// TwinCAT 3 PLC project Temp_PID_cascade
// ProgramVersion: 3.1.4023.0
// libraries:
//   Tc2_ControllerToolbox,3.4.1.4,Beckhoff Automation GmbH
//   Tc2_Math,3.3.1.0,Beckhoff Automation GmbH
//   Tc2_Standard,3.3.3.0,Beckhoff Automation GmbH
//   Tc2_System,3.4.22.0,Beckhoff Automation GmbH
//   Tc2_TempController,3.3.4.0,Beckhoff Automation GmbH
//   Tc3_Module,3.3.21.0,Beckhoff Automation GmbH
// project tree:
//   GVLs/ gbl.TcGVL, IOgbl.TcGVL
//   / PlcTask.TcTTO
//   POUs/ MAIN.TcPOU, master.TcPOU, slave.TcPOU
// real-time tasks:
//   TASK PlcTask: cycle T#1ms, priority 20, ADS port 350
// I/O:
//   DEVICE Device 1 (EtherCAT) (disabled), AmsNetId 192.168.56.1.2.1
//     Term 1 (EK1200) [EK1200-5000 EtherCAT Power supply (2A E-Bus)]
//       Term 2 (EL3318) [EL3318 8Ch. Ana Input Thermocouple (TC)]
//       Term 3 (EL3318) [EL3318 8Ch. Ana Input Thermocouple (TC)]
//       Term 4 (EL4024) [EL4024 4Ch. Ana. Output 4-20mA, 12bit]
//       Term 5 (EL9011) [EL9011 End Terminal]
// variable links:
//   Temp_PID_cascade/Temp_PID_cascade Instance <-> Device 1 (EtherCAT)/Term 1 (EK1200)/Term 2 (EL3318)
//     PlcTask Inputs/IOgbl.AI_IO_ST_temp[1] <-> TC Channel 8/Value
//     PlcTask Inputs/IOgbl.AI_IO_slave_pv[{1..4}] <-> TC Channel {1..4}/Value  (4 links)
//   Temp_PID_cascade/Temp_PID_cascade Instance <-> Device 1 (EtherCAT)/Term 1 (EK1200)/Term 3 (EL3318)
//     PlcTask Inputs/IOgbl.AI_IO_ST_temp[{2..9}] <-> TC Channel {1..8}/Value  (8 links)
//   Temp_PID_cascade/Temp_PID_cascade Instance <-> Device 1 (EtherCAT)/Term 1 (EK1200)/Term 4 (EL4024)
//     PlcTask Outputs/IOgbl.AO_IO_SCR_set[{1..4}] <-> AO Outputs Channel {1..4}/Analog output  (4 links)

CONFIGURATION Temp_PID_cascade
    RESOURCE PLC ON TwinCAT3
        TASK PlcTask(INTERVAL := T#1ms, PRIORITY := 20);
        PROGRAM MAIN WITH PlcTask : MAIN;
    END_RESOURCE
END_CONFIGURATION

// ---- GVLs/gbl.TcGVL
{attribute 'qualified_only'}
VAR_GLOBAL
	(*===========================================main=====================================*)
	bWatch						 : BOOL;
	tuning_mode 	     		 : BOOL;
	tuning_time	     			 : LREAL;
	tune_result					 :  ARRAY[1..4] OF LREAL;
	
	(*===========================================master====================================*)
	master_bRamp_Enable          : BOOL;
	(*---------------------input------------------------*)
	master_fRamp_Value           : ARRAY[1..4] OF LREAL := [10, 10, 10, 10] ;
	master_TargetTemp            : LREAL;
	master_pi_gain               : ARRAY[1..4] OF LREAL;	//PI제어기 이득(gain) -P
	master_integral_constant	 : ARRAY[1..4] OF LREAL;	//PI제어기 적분상수 -I
	master_Zone_Temp_Min         : LREAL;  //단위 : %
	master_Zone_Temp_Max         : LREAL;  //단위 : %
	
	(*===========================================sub TC===================================*)
	(*---------------------output------------------------*)
	fPV_Value_SubTC				: ARRAY[1..9] OF LREAL; (* glass 각각의 온도 *)
	subTC_max 					: LREAL ;
	subTC_min 					: LREAL ;
	subTC_dev					: LREAL ;  (* glss_max - glass_min *)
	subTC_AVG                   : LREAL ;  (* glass temp AVG *)
	
	(*=======================================slave========================================*)	
	slave_bsimulation		   : BOOL;
	slave_bRamp_Enable         : ARRAY[1..4] OF BOOL;
	(*---------------------input------------------------*)
	slave_fRamp_Value          : ARRAY[1..4] OF LREAL ;
	slave_fTargetTemp          : ARRAY[1..4] OF LREAL ;
	slave_fPowLimit            : ARRAY[1..4] OF LREAL ;
	slave_eCTRL_MODE           : ARRAY[1..4] OF E_CTRL_MODE ;
	slave_bstart			   : BOOL ;

	slave_fP_Value	           : ARRAY[1..4] OF LREAL  ;
	slave_tI_Value		       : ARRAY[1..4] OF LREAL  ;
	slave_tD_Value		       : ARRAY[1..4] OF LREAL  ;
	slave_bEmergency_Stop	   : BOOL ;
	(*---------------------output------------------------*)
	slave_fPV_Value				: ARRAY[1..4] OF LREAL;
	slave_fMV_Out				: ARRAY[1..4] OF LREAL;
	slave_fRamp_Out 		    : ARRAY[1..4] OF LREAL;
	slave_nErrorID			    : E_CTRL_ERRORCODES;	
	slave_bError				: BOOL;
END_VAR

// ---- GVLs/IOgbl.TcGVL
{attribute 'qualified_only'}
VAR_GLOBAL
	AI_IO_slave_pv  AT%IB1001   :   ARRAY [1..4] OF UINT;
	AI_IO_ST_temp   AT%IB1021   :   ARRAY [1..9] OF UINT;
	
	
	AO_IO_SCR_set 	AT%QB1051 	:   ARRAY [1..4] OF UINT;  
END_VAR

// ---- POUs/MAIN.TcPOU
PROGRAM MAIN
VAR	
	onTimer 			: TON;
	OffTimer 			: TOF;
	timerStart			: BOOL;
	reverseSignal 		: BOOL;
	
	onTimer_tune  		: TON;
	OffTimer_tune 		: TOF;
	reverseSignal_tune  : BOOL;
	
	i    				: INT;

END_VAR


IF gbl.slave_bsimulation = FALSE THEN

	FOR i:=1 TO 4 BY 1 DO
		gbl.slave_fPV_Value[i] := IOgbl.AI_IO_slave_pv[i] / 10 ;
		IOgbl.AO_IO_SCR_set[i] := LREAL_TO_UINT(gbl.slave_fMV_Out[i] * 327.67);
	END_FOR
	
	FOR i:=1 TO 9 BY 1 DO
		gbl.fPV_Value_SubTC[i] := IOgbl.AI_IO_ST_temp[i] / 10 ;
	END_FOR
	
ELSE
	slave.SIMULATION() ;
END_IF

(* watch dogs : 10s 간격으로 on/ off *)
onTimer(IN := OffTimer.Q, PT := T#10S);
IF onTimer.Q THEN
  reverseSignal := FALSE;
  gbl.bWatch := FALSE;
ELSE
  reverseSignal := TRUE;
  gbl.bWatch := TRUE;
END_IF
OffTimer(IN := reverseSignal, PT := T#10S);

(* 
mgbl.master_tuning_mode = tune set
tune set :  true -> master, slave호출
tune set :  false -> slave만 호출
*)
IF gbl.tuning_mode THEN

	master();
	slave();
	
  (* 튜닝 시간 설정 = mgbl.master_tuning_time *)
    onTimer_tune(IN := OffTimer_tune.Q, PT := LREAL_TO_TIME(gbl.tuning_time)*60000); // IN이 FALSE에서 TRUE가 되자마자 시간이 흐름,PT와 같아지면 Q가 TRUE
    IF onTimer_tune.Q THEN
	  gbl.tuning_mode := FALSE;
	  reverseSignal_tune := FALSE;
	  gbl.tune_result := gbl.slave_fPV_Value;
	ELSE
	  reverseSignal_tune := TRUE;
    END_IF
    OffTimer_tune(IN := reverseSignal_tune, PT := T#0S); // IN이 TRUE에서 FALSE가 되자마자 시간이 흐름, PT와 같아지면 Q가 FALSE
	FOR i:=1 TO 4 BY 1 DO
		gbl.tune_result[i] := 0;
	END_FOR
ELSE
	slave();
END_IF

END_PROGRAM

// ---- POUs/slave.TcPOU
PROGRAM slave
VAR
	fPV_Value_					:			ARRAY[1..4] OF LREAL ;
	
	tTime						:			TIME ;
	tTaskCycleTime				:			TIME := T#1MS ;
	tCtrlCycleTime				:			TIME := T#200MS ;
	
	fbCTRL_PT2				    : 			ARRAY[1..4] OF FB_CTRL_PT2 ;
	stPTParams				    : 			ARRAY[1..4] OF ST_CTRL_PT2_PARAMS ;

	stCTRL_ParaController_Ex	:			ARRAY[1..4] OF ST_CTRL_ParaController ;
	stCTRL_ParaController_In	:			ARRAY[1..4] OF ST_CTRL_ParaController ;
	stCTRL_TempCtrlParameter	:			ARRAY[1..4] OF ST_CTRL_TempCtrlParameter ;
	
	fbCTRL_TempController		:			ARRAY[1..4] OF FB_CTRL_TempController ;
		
	eCTRL_STATE					:			ARRAY[1..4] OF E_CTRL_STATE ;
	
	e_Heat_Mode					:			E_CTRL_ControlMode 			:= eCTRL_ControlMode_HEATING ;
	e_Fail_Action				:			E_CTRL_ReactionOnFailure 	:= eCTRL_ReactionOnFailure_NoFailure ;
		
	s_bError					:			BOOL ;
	s_nErrorID					:			E_CTRL_ERRORCODES ;
	s_fMaxOvershoot				:			LREAL ;
	
	s_bFirst					:			BOOL := TRUE ;
	
	(* Ramp Parameter Set *)
	s_bRamp_Use				    :			ARRAY[1..4] OF BOOL ;	
	s_fRamp_Rate				:			ARRAY[1..4] OF LREAL ;
	
	(* =============== Setting Item 입력 =============== *)
	
	(* PID Set Parameter *)
	s_fP_Value						:			ARRAY[1..4] OF LREAL ;
	s_tI_Value						:			ARRAY[1..4] OF TIME	;
	s_tD_Value						:			ARRAY[1..4] OF TIME	;
	
	(* Power Limit Set *)
	s_fPowLimit					:			ARRAY[1..4] OF LREAL ;
	
	(* Manual Control 시 Power 출력값 *)
	s_fSetManual					:			ARRAY[1..4] OF LREAL ;
	
	(*	Heater Mode	*)
	s_eCTRL_MODE					:			ARRAY[1..4] OF E_CTRL_MODE ;			(* Auto Mode 동작은 2 : eCTRL_MODE_ACTIVE 설정 *)
	
	(*	온도 설정 입력	*)
	s_fSet_Value					:			ARRAY[1..4] OF LREAL ;
	s_fLast_Set_Value            	:           ARRAY[1..4] OF LREAL ;

	
	(*	비상정지	*)
	//bEmergency_Stop					:			ARRAY[1..4] OF BOOL ;
	
	fbCTRL_RAMP_GENERATOR			 :   ARRAY[1..4] OF FB_CTRL_RAMP_GENERATOR ;
	stCTRL_RAMP_GENERATOR_PARAMS     :   ARRAY[1..4] OF ST_CTRL_RAMP_GENERATOR_PARAMS ;
	
	System_step	: INT ;
	
	i    :   INT ;
	
	master_Zone_AVG	                 :   ARRAY[1..4] OF LREAL ;
	
END_VAR

(* ================ Simulation Constant Parameter =======================*)
VAR CONSTANT
	fKp							:			ARRAY[1..4] OF REAL := [15.5, 15.2, 15.7, 15.8] ;
	fInit_Temp					:			ARRAY[1..4] OF REAL := [23.5, 23.8, 23.9, 23.7] ;
	tTimeConstant				:			ARRAY[1..4] OF TIME := [T#251.4S, T#252.4S, T#254.4S, T#256.4S] ;
END_VAR

(*
IF gbl.slave_bsimulation THEN
   SIMULATION();
END_IF
*)

IF gbl.slave_bError THEN
   gbl.slave_bEmergency_Stop := TRUE ;
END_IF

FOR i:=1 TO 4 BY 1 DO
   IF gbl.slave_bEmergency_Stop THEN
      s_fSet_Value[i] := 0;
      s_fPowLimit[i] := 0;
      s_eCTRL_MODE[i] := eCTRL_MODE_IDLE;
      fbCTRL_TempController[i]( eCtrlMode := s_eCTRL_MODE[i],      
              bSelSetpoint            := FALSE,
              fw1                     := s_fSet_Value[i],
              fw2                     := ,            
              fX                      := gbl.slave_fPV_Value[i],      
              fyManual                := s_fSetManual[i],
              sParaControllerExternal := stCTRL_ParaController_Ex[i],
              sControllerParameter    := stCTRL_TempCtrlParameter[i]
              );
   ELSE
      s_fPowLimit[i] := gbl.slave_fPowLimit[i];
      s_eCTRL_MODE[i] := gbl.slave_eCTRL_MODE[i];
   END_IF
END_FOR

IF s_bFirst THEN
   DEFAULT_PARA_SET();
   s_bFirst := FALSE ;
   System_step :=0;
END_IF

CASE System_step OF
      
   0:

      s_bRamp_Use     :=  gbl.slave_bRamp_Enable;
      s_fRamp_Rate    :=  gbl.slave_fRamp_Value;
	  
      IF gbl.slave_bStart THEN
         FOR i:=1 TO 4 BY 1 DO
            s_fLast_Set_Value[i] := s_fSet_Value[i];
         END_FOR
         FOR i:=1 TO 4 BY 1 DO
            s_fSet_Value[i] := gbl.slave_fTargetTemp[i];
         END_FOR
         System_step := 1;
         gbl.slave_bStart := FALSE;
         ELSE
            System_step := 0;
      END_IF
      

   1:
      FOR i:=1 TO 4 BY 1 DO
         s_fP_Value[i] := gbl.slave_fP_Value[i];
         s_tI_Value[i] := LREAL_TO_TIME(gbl.slave_tI_Value[i]);
         s_tD_Value[i] := LREAL_TO_TIME(gbl.slave_tD_Value[i]);
         
         IF s_fP_Value[i] <= 0 THEN
            s_fP_Value[i] := 0.1;
         ELSE
            s_fP_Value[i] := s_fP_Value[i];
         END_IF

         stCTRL_ParaController_Ex[i].KpHeat := s_fP_Value[i];   
         stCTRL_ParaController_Ex[i].TnHeat := s_tI_Value[i];
         stCTRL_ParaController_Ex[i].TvHeat := s_tD_Value[i];
         stCTRL_ParaController_Ex[i].TdHeat := T#1S;
         
         System_step := 2;
         
      END_FOR
      
      System_step := 2;

   2:
      
      FOR i:=1 TO 4 BY 1 DO
         IF s_fPowLimit[i] > 100 THEN
            s_fPowLimit[i] := 100;
         ELSE 
            s_fPowLimit[i] := s_fPowLimit[i];
         END_IF
      
         stCTRL_TempCtrlParameter[i].fYMax := s_fPowLimit[i];
         
         stCTRL_RAMP_GENERATOR_PARAMS[i].fVeloNeg := s_fRamp_Rate[i] / 60.0;
         stCTRL_RAMP_GENERATOR_PARAMS[i].fVeloPos := s_fRamp_Rate[i] / 60.0;
         
         System_step := 3;
      
      END_FOR
       
      System_step := 3;
   
   3:
      
      FOR i:=1 TO 4 BY 1 DO
      
         IF s_fSetManual[i] > 100 THEN
            s_fSetManual[i] := 100;
         ELSE
            s_fSetManual := s_fSetManual;
         END_IF

         stCTRL_TempCtrlParameter[i].fYManual         :=   s_fSetManual[i];          
         stCTRL_TempCtrlParameter[i].fYOnFailure      :=   s_fSet_Value[i];
      END_FOR
      
      System_step := 4;
     
   4:
      FOR i:=1 TO 4 BY 1 DO
         fbCTRL_TempController[i]( eCtrlMode               := gbl.slave_eCTRL_MODE[i],      
                             bSelSetpoint            := FALSE,
                             fw1                     := s_fSet_Value[i],
                             fw2                     := ,            
                             fX                      := gbl.slave_fPV_Value[i],      
                             fyManual                := s_fSetManual[i],
                             sParaControllerExternal := stCTRL_ParaController_Ex[i],
                             sControllerParameter    := stCTRL_TempCtrlParameter[i]
                             );
        END_FOR
      
      System_step := 100;
      
   100:
      System_step := 0;
      
END_CASE


Ramping();

FOR i:=1 TO 4 BY 1 DO 
   
   fbCTRL_TempController[i](
                 fw1                       := gbl.slave_fRamp_Out[i],
                 fX                        := gbl.slave_fPV_Value[i],    
                 sParaControllerExternal   := stCTRL_ParaController_Ex[i],
                 sControllerParameter      := stCTRL_TempCtrlParameter[i],
                 fYAnalog                   => gbl.slave_fMV_Out[i],
                 bYPWMPos                   => ,
                 bYPWMNeg                   => ,
                 dwAlarm                    => ,
                 fMaxOverShoot              => s_fMaxOvershoot,
                 tStartUpTime               => ,
                 eCtrlState                 => eCTRL_STATE[i],
                 sParaControllerInternal    => stCTRL_ParaController_In[i],
                 bError                     => gbl.slave_bError,
                 eErrorId                   => gbl.slave_nErrorID
                );
END_FOR

ACTION DEFAULT_PARA_SET:
FOR i := 1 TO 4 DO
	stCTRL_TempCtrlParameter[i].iMode				:=	e_Heat_Mode;
	stCTRL_TempCtrlParameter[i].iReactionOnFailure  :=	e_Fail_Action;
	stCTRL_TempCtrlParameter[i].dwAlarmSupp		    :=	16#FF_FF_FF_FF;		(* alarm suppression  Default 사용 *)
	stCTRL_TempCtrlParameter[i].fWMin				:=	0.0;
	stCTRL_TempCtrlParameter[i].fWMax				:=	500;
	stCTRL_TempCtrlParameter[i].bEnableSoftStart	:=	FALSE;
	stCTRL_TempCtrlParameter[i].fWStartUp			:=	30.0;
	stCTRL_TempCtrlParameter[i].tStartUp			:=	T#1S;
	stCTRL_TempCtrlParameter[i].bStartUpRamping	    :=	FALSE;
	stCTRL_TempCtrlParameter[i].fWStartUpVeloPos	:=	0.1;
	stCTRL_TempCtrlParameter[i].fWStartUpVeloNeg	:=	0.1;
	stCTRL_TempCtrlParameter[i].bFilter			    :=	FALSE;
	stCTRL_TempCtrlParameter[i].tFilter			    :=	T#0S;
	stCTRL_TempCtrlParameter[i].bDeadband			:=	FALSE;
	stCTRL_TempCtrlParameter[i].fEDeadband			:=	0.0;
	stCTRL_TempCtrlParameter[i].tPWMCycleTime		:=	T#1S;
	stCTRL_TempCtrlParameter[i].tPWMMinOffTime		:=	T#0S;
	stCTRL_TempCtrlParameter[i].tPWMMinOnTime		:=	T#0S;
	stCTRL_TempCtrlParameter[i].tPWMWaitingTime	    :=	T#0S;
	stCTRL_TempCtrlParameter[i].fYThresholdOff		:=	0.0;
	stCTRL_TempCtrlParameter[i].fYThresholdOn		:=	0.0;
	stCTRL_TempCtrlParameter[i].TempLow			    :=	-10.0;
	stCTRL_TempCtrlParameter[i].TempLowLow			:=	-5.0;
	stCTRL_TempCtrlParameter[i].TempHigh			:=	5.0;
	stCTRL_TempCtrlParameter[i].TempHighHigh		:=	10.0;
	stCTRL_TempCtrlParameter[i].TempAbsoluteHigh	:=	300.0;
	stCTRL_TempCtrlParameter[i].TempAbsoluteLow	    :=	0.0;
	stCTRL_TempCtrlParameter[i].tCtrlCycleTime		:= 	tCtrlCycleTime;
	stCTRL_TempCtrlParameter[i].tTaskCycleTime		:= 	tTaskCycleTime;
	stCTRL_TempCtrlParameter[i].fYMin				:=	0.0;
	stCTRL_TempCtrlParameter[i].iControllerType	    := eCTRL_ControllerType_PID;
	stCTRL_TempCtrlParameter[i].iFilterType		    := eCTRL_FilterType_FIRSTORDER;
	stCTRL_TempCtrlParameter[i].bEnablePreController:= FALSE;
	stCTRL_TempCtrlParameter[i].bEnableZones 		:= FALSE;
	stCTRL_TempCtrlParameter[i].bEnableCVFilter     := FALSE;
	
	stCTRL_TempCtrlParameter[i].bSelCtrlParameterSet := TRUE;
	
	stCTRL_RAMP_GENERATOR_PARAMS[i].tCtrlCycleTime		:= 	tCtrlCycleTime;
	stCTRL_RAMP_GENERATOR_PARAMS[i].tTaskCycleTime		:= 	tTaskCycleTime;
END_FOR
END_ACTION

ACTION RAMPING:

;
FOR i:=1 TO 4 BY 1 DO
	IF s_bRamp_Use[i] THEN

		fbCTRL_RAMP_GENERATOR[i]( bEnable   := s_bRamp_Use[i],
								fStart   := s_fLast_Set_Value[i],
								fTarget  := s_fSet_Value[i],
								stParams := stCTRL_RAMP_GENERATOR_PARAMS[i],
								fOut   => gbl.slave_fRamp_Out[i],
								fVeloOut  => ,
								bValueReached => ,
								eErrorId => ,
								bError =>
								)
	;			

	ELSE
			gbl.slave_fRamp_Out[i] := s_fSet_Value[i];
		;
	END_IF
END_FOR
END_ACTION

ACTION SIMULATION:


FOR i:=1 TO 4 BY 1 DO
	stPTParams[i].tTaskCycleTime	:= tTaskCycleTime;
	stPTParams[i].tCtrlCycleTime	:= tCtrlCycleTime;
	stPTParams[i].tT1				:= stPTParams[i].tT2 := tTimeConstant[i];
	stPTParams[i].fKp				:= fKp[i];


	fbCTRL_PT2[i](
					fIn			:= gbl.slave_fMV_Out[i] ,
					eMode		:= eCtrl_MODE_ACTIVE,
					stParams	:= stPTParams[i],
					fOut		=> fPV_Value_[i]
					);	
					
	IF fPV_Value_[i] <= fInit_Temp[i] THEN
		gbl.slave_fPV_Value[i] := fInit_Temp[i];
	ELSE
		gbl.slave_fPV_Value[i] := fPV_Value_[i];
	END_IF 	
	
END_FOR
END_ACTION

END_PROGRAM

// ---- POUs/master.TcPOU
PROGRAM master
VAR
(*-------------------------------------------- master 입력 변수 --------------------------------------------*)	
	m_bRamp_Enable                   : BOOL;
	m_fRamp_Value                    : ARRAY[1..4] OF LREAL;
	
	m_fTargetTemp                    : LREAL;
	m_btuning_mode 	     			 : BOOL;
	m_Sampling_Time					 : LREAL := 10;             // Sampling time (적용시간 간격  Δt(*고정값*))
	m_integral_constant			 	 : ARRAY[1..4] OF LREAL;	//PI제어기 적분상수
	m_pi_gain                        : ARRAY[1..4] OF LREAL;	//PI제어기 이득(gain)
	
	m_Set_Value						 : ARRAY[1..4] OF LREAL;
	m_fLast_Set_Value            	 : ARRAY[1..4] OF LREAL;
	m_Heatup_On				 		 : BOOL;
	m_Tuning_Set_Temp				 : ARRAY[1..4] OF LREAL;
	m_Tuning_Set_Temp_Sum			 : LREAL;
	m_Tuning_Set_Temp_Avg			 : LREAL;
	m_Tune_On						 : BOOL;
	bStart							 : BOOL;
	bSecondStart					 : BOOL;
	bThirdStart						 : BOOL;
	m_Heatup_Start_Temp				 : ARRAY[1..4] OF LREAL;
	m_Heatup_End_Temp				 : ARRAY[1..4] OF LREAL;
	m_Heatup_Start_Temp_Sum			 : LREAL;
	m_Heatup_Start_Temp_Avg			 : LREAL;
	m_Zone_Sum						 : LREAL;
	m_Zone_Avg						 : LREAL; // ActTemp(fPV_Value) 평균
	m_Zone_Max						 : LREAL;
	m_Zone_Min						 : LREAL;
	m_Zone_Dev						 : LREAL;
	
	tWait_Time						 :	TON;
(*---------------------------------------- Substrate Simulation ----------------------------------------------- *)
	fMV_Out						     : ARRAY[1..4] OF LREAL;
	fMV_Out_Sub					     : ARRAY[1..9] OF LREAL;
	fPV_Value_Sub					 : ARRAY[1..9] OF LREAL;
	fPV_Value_Local_Sub				 : ARRAY[1..9] OF LREAL;
	fbCTRL_PT2_Sub			         : ARRAY[1..9] OF FB_CTRL_PT2;
	stPTParams_Sub			         : ARRAY[1..9] OF ST_CTRL_PT2_PARAMS;
	fKp_Sub						     : ARRAY[1..9] OF REAL := [15.7, 15.8, 15.3, 15.1, 15.0, 15.5, 15.6, 15.2, 15.4];
	fInit_Temp_Sub				     : ARRAY[1..9] OF REAL := [23.5, 23.6, 23.7, 23.8, 23.9, 24.0, 24.1, 24.2, 24.3];
	tTimeConstant_Sub			     : ARRAY[1..9] OF TIME := [T#325.7S, T#335.5S, T#328.4S, T#321.9S, T#330.3S, T#324.2S, T#329.9S, T#329.4S, T#325.1S];
	
(*-------------------------------------------- master 출력 변수 --------------------------------------------*)

	master_Zone_AVG                :   ARRAY[1..4] OF LREAL;                	// 글래스 온도 평균(4개 더해서 4로 나눔)
	master_subTC 				   :   LREAL;
	
	Substrate_AvgTemp			   :   ARRAY[1..4] OF LREAL;
	
	mErr_Value                     :   ARRAY[1..4] OF LREAL;                    // 제어오차 (set_temp - msater_subTC_AVG)
	mErr_integral_Val			   :   ARRAY[1..4] OF LREAL := [0 , 0, 0, 0 ];  // 오차의 적분(se , 초기값 = 0)
	
	m_min_per					   :	LREAL;
	m_max_per					   :	LREAL;
	m_Zone_Temp_Min                :    LREAL;
	m_Zone_Temp_Max                :    LREAL;
	
	m_Last_Zone_Temp_AVG		   :	ARRAY[1..4] OF LREAL; 
	
	i							   :	INT;
	j							   : 	INT;
	
	fbCTRL_RAMP_GENERATOR		   :    ARRAY[1..4] OF FB_CTRL_RAMP_GENERATOR;
	stCTRL_RAMP_GENERATOR_PARAMS   :    ARRAY[1..4] OF ST_CTRL_RAMP_GENERATOR_PARAMS;
	
	tTime						   :	TIME;
	tTaskCycleTime				   :	TIME := T#1MS;
	tCtrlCycleTime				   :	TIME := T#200MS;
	
	fbCTRL_PT2				       : 	ARRAY[1..4] OF FB_CTRL_PT2;
	stPTParams				       : 	ARRAY[1..4] OF ST_CTRL_PT2_PARAMS;
	
	glass_max 					   :	LREAL ;
	glass_min 					   :	LREAL ;
	glass_dev					   :	LREAL ;       (* glss_max - glass_min *)
	glass_AVG                      : 	LREAL;        (* 글래스 온도 평균(9개 평균 = g_bar)*)
	
	mErr_Old_Value                 :   	ARRAY[1..4] OF LREAL;   (* 전회 제어 오차 *)
	fKd							   : 	LREAL := 1;		(* 공정 상수 *)
	
(*===================================결과 출력값==========================================================*)
	result_zone_set_val			   :	ARRAY [1..4] OF LREAL ;
	result_glass_dev			   :	LREAL := 10 ;
	result_subTC_AVG			   :	LREAL := 0 ;
	rampBool 					   :	BOOL ;
	zoneIndex					   :	INT ;
	
(* ------------------------------------------Ramp Parameter Set-------------------------------------- *)
	m_bRamp_Use				       :	BOOL ;	
	m_fRamp_Rate				   :	ARRAY[1..4] OF LREAL := [10 , 10, 10 , 10 ];
	m_fRamp_Out 			       : 	ARRAY[1..4] OF LREAL ;	
	
END_VAR

Substrate_AVG();

IF gbl.bTimeOver THEN
	m_Tune_On := FALSE;
	bStart := FALSE;
	m_Heatup_On := FALSE;
	bSecondStart := FALSE;
	bThirdStart := FALSE;
	gbl.slave_bstart := TRUE;
END_IF

m_integral_constant  := gbl.master_integral_constant;
m_pi_gain    		 := gbl.master_pi_gain;
m_fTargetTemp		 := gbl.master_TargetTemp;
m_min_per		     := gbl.master_Zone_Temp_Min;
m_max_per	         := gbl.master_Zone_Temp_Max;
fPV_Value_Sub   	 := gbl.fPV_Value_SubTC ;
gbl.subTC_max		 := glass_max ;
gbl.subTC_min		 := glass_min ;
gbl.subTC_dev		 := glass_dev ;
gbl.subTC_AVG		 := glass_AVG ;
master_subTC 		 := 0 ;
tWait_Time(IN := TRUE, PT := LREAL_TO_TIME(m_Sampling_Time) * 1000);

glass_max := 0;
glass_min := 1000;
master_subTC := 0;
m_Zone_Max := 0;
m_Zone_Min := 1000;
m_Zone_Dev := 0;

FOR i:=1 TO 9 BY 1 DO
	master_subTC := master_subTC + gbl.fPV_Value_SubTC[i];
	glass_max := MAX(glass_max, gbl.fPV_Value_SubTC[i]);
	glass_min := MIN(glass_min, gbl.fPV_Value_SubTC[i]);
END_FOR
glass_dev := glass_max - glass_min;	
glass_AVG := master_subTC /9;

IF glass_dev <= 10 THEN
	IF result_glass_dev > glass_dev THEN
		result_glass_dev := glass_dev;
	END_IF
	
	IF (m_fTargetTemp * 0.9) <= glass_AVG AND (m_fTargetTemp * 1.1) >= glass_AVG THEN
		IF ABS(m_fTargetTemp - glass_AVG) < ABS(m_fTargetTemp - result_subTC_AVG) THEN
			result_subTC_AVG := glass_AVG;
		END_IF
	END_IF
END_IF

IF gbl.slave_bstart THEN
	IF gbl.tuningIndex=0 THEN
		m_Zone_Sum := 0;
		FOR i:=1 TO 4 BY 1 DO
			m_Zone_Sum := m_Zone_Sum + gbl.slave_fPV_Value[i];
		END_FOR
		m_Zone_Avg := m_Zone_Sum / 4;
		FOR i:=1 TO 4 BY 1 DO
			m_Tuning_Set_Temp[i] := m_Zone_Avg;
		END_FOR
	ELSE
		m_Tuning_Set_Temp := m_Heatup_Start_Temp;
	END_IF
	m_Tuning_Set_Temp_Sum := 0;
	FOR i:=1 TO 4 BY 1 DO
		m_Tuning_Set_Temp_Sum := m_Tuning_Set_Temp_Sum + m_Tuning_Set_Temp[i];
	END_FOR
	m_Tuning_Set_Temp_Avg := m_Tuning_Set_Temp_Sum / 4;
	m_Zone_Temp_Min := m_Tuning_Set_Temp_Avg - (m_Tuning_Set_Temp_Avg * m_min_per / 100);
	m_Zone_Temp_Max := m_Tuning_Set_Temp_Avg + (m_Tuning_Set_Temp_Avg * m_max_per / 100);
	FOR i:=1 TO 4 BY 1 DO
		mErr_integral_Val[i] := 0;
	END_FOR
	m_tune_On := TRUE;
	bStart := TRUE;
END_IF

IF m_Tune_On THEN
	IF tWait_Time.Q THEN
		tWait_Time(IN := FALSE);
		Tuning();
	END_IF
END_IF

FOR i:=1 TO 4 BY 1 DO
	m_Zone_Max := MAX(m_Zone_Max, gbl.slave_fPV_Value[i]);
	m_Zone_Min := MIN(m_Zone_Min, gbl.slave_fPV_Value[i]);
END_FOR
m_Zone_Dev := m_Zone_Max - m_Zone_Min;

IF bStart THEN
	IF glass_dev <= 2.5 THEN
		m_Heatup_On := TRUE;
		m_Tune_On := FALSE;
		IF gbl.tuningIndex=0 THEN
			m_Heatup_Start_Temp := gbl.slave_fPV_Value;
		END_IF
		bSecondStart := TRUE;
		bStart := FALSE;
		gbl.isChanged := TRUE;
		FOR i:=1 TO 4 BY 1 DO
			gbl.slave_fTargetTemp[i] := gbl.master_TargetTemp;
		END_FOR
		FOR i:=1 TO 4 BY 1 DO
			FOR j:=1 TO gbl.arrSize BY 1 DO
				gbl.newData[i, j] := 0;
			END_FOR
		END_FOR
	END_IF
END_IF

IF m_Heatup_On THEN
	m_Zone_Temp_Min := gbl.master_TargetTemp - (gbl.master_TargetTemp * m_min_per / 100);
	m_Zone_Temp_Max := gbl.master_TargetTemp + (gbl.master_TargetTemp * m_max_per / 100);
	IF tWait_Time.Q THEN
		tWait_Time(IN := FALSE);
		HEATUP();
	END_IF
END_IF

IF bSecondStart THEN
	IF gbl.master_TargetTemp <= glass_AVG THEN
		IF gbl.tuningIndex=0 THEN			
			FOR i:=1 TO 4 BY 1 DO
				m_Tuning_Set_Temp[i] := gbl.master_TargetTemp;
			END_FOR
		ELSE
			m_Tuning_Set_Temp := m_Heatup_End_Temp;
		END_IF
		m_Tuning_Set_Temp_Sum := 0;
		FOR i:=1 TO 4 BY 1 DO
			m_Tuning_Set_Temp_Sum := m_Tuning_Set_Temp_Sum + m_Tuning_Set_Temp[i];
		END_FOR
		m_Tuning_Set_Temp_Avg := m_Tuning_Set_Temp_Sum / 4;
		m_Zone_Temp_Min := m_Tuning_Set_Temp_Avg - (m_Tuning_Set_Temp_Avg * m_min_per / 100);
		m_Zone_Temp_Max := m_Tuning_Set_Temp_Avg + (m_Tuning_Set_Temp_Avg * m_max_per / 100);
		m_Tune_On := TRUE;
		m_Heatup_On := FALSE;
		bThirdStart := TRUE;
		bSecondStart := FALSE;
	END_IF
END_IF

IF bThirdStart THEN
	IF glass_dev <= 2.5 THEN
		m_Tune_On := FALSE;
		bThirdStart := FALSE;
		IF gbl.tuningIndex = (gbl.tuningCount-1) THEN
			gbl.tuningIndex := 0;
			gbl.tuning_mode := FALSE;
			gbl.heatupData[gbl.tuningCount + 1 - gbl.tuningIndex - 1] 	:= gbl.newData;
			RETURN;
		END_IF
		gbl.isDropping := TRUE;
		gbl.isChanged := TRUE;
		IF gbl.tuningIndex=0 THEN
			m_Heatup_End_Temp := gbl.slave_fPV_Value;
		END_IF
		gbl.slave_fTargetTemp := m_Heatup_Start_Temp;
	END_IF
END_IF

m_Heatup_Start_Temp_Sum := 0;
FOR i:=1 TO 4 BY 1 DO
	m_Heatup_Start_Temp_Sum := m_Heatup_Start_Temp_Sum + m_Heatup_Start_Temp[i];
END_FOR
m_Heatup_Start_Temp_Avg := m_Heatup_Start_Temp_Sum / 4;

IF gbl.isDropping THEN
	IF glass_AVG <= m_Heatup_Start_Temp_Avg THEN
		gbl.bRestart := TRUE;
		gbl.tuningIndex := gbl.tuningIndex + 1;
		gbl.index := 1;
		gbl.isDropping := FALSE;
	END_IF
END_IF

ACTION HEATUP:
(*
m_bRamp_Use     :=  gbl.master_bRamp_Enable := TRUE;
m_fRamp_Rate    :=  gbl.master_fRamp_Value;
FOR i:=1 TO 4 BY 1 DO
	stCTRL_RAMP_GENERATOR_PARAMS[i].fVeloNeg := m_fRamp_Rate[i] / 60.0;
	stCTRL_RAMP_GENERATOR_PARAMS[i].fVeloPos := m_fRamp_Rate[i] / 60.0;
END_FOR

IF m_bRamp_Use THEN
	FOR i:=1 TO 4 BY 1 DO
		fbCTRL_RAMP_GENERATOR[i]( bEnable   := m_bRamp_Use,
								fStart  	:= m_Heatup_Start_Temp[i],
								fTarget 	:= m_fTargetTemp,
								stParams    := stCTRL_RAMP_GENERATOR_PARAMS[i],
								fOut    	 => m_fRamp_Out[i],
								fVeloOut  	 => ,
								bValueReached => ,
								eErrorId => ,
								bError =>
								)
	;
	END_FOR					

ELSE
	FOR i:=1 TO 4 BY 1 DO
		m_fRamp_Out[i] := m_fTargetTemp;
	;
	END_FOR
END_IF
*)
IF gbl.tuningIndex=0 THEN
	FOR i:=1 TO 4 BY 1 DO
		gbl.slave_fTargetTemp[i] := gbl.master_TargetTemp;
		master_Zone_AVG[i] := gbl.slave_fPV_Value[i];
	END_FOR
END_IF

(* tuning data 저장 *)
FOR zoneIndex:=1 TO 4 BY 1 DO
	IF gbl.tuningIndex <> 0 THEN
		master_Zone_AVG[zoneIndex] := gbl.oldData[zoneIndex, gbl.index] + fKd * ( mErr_Value[zoneIndex] - mErr_Old_Value[zoneIndex]);
		mErr_Old_Value[zoneIndex]  := mErr_Value[zoneIndex] ;
		IF gbl.heatupData[gbl.tuningCount + 1 - gbl.tuningIndex][zoneIndex, gbl.index]=0 THEN
			continue;
		END_IF
		gbl.slave_fTargetTemp[zoneIndex] := gbl.heatupData[gbl.tuningCount + 1 - gbl.tuningIndex][zoneIndex, gbl.index];
		gbl.isChanged := TRUE;
	END_IF
	gbl.newData[zoneIndex, gbl.index] := master_Zone_AVG[zoneIndex];
END_FOR
gbl.index := gbl.index + 1 ;
END_ACTION

ACTION Substrate_AVG:
Substrate_AvgTemp[1] := (fPV_Value_Sub[1] + fPV_Value_Sub[2] + fPV_Value_Sub[4] + fPV_Value_Sub[5]) / 4; 
Substrate_AvgTemp[2] := (fPV_Value_Sub[2] + fPV_Value_Sub[3] + fPV_Value_Sub[5] + fPV_Value_Sub[6]) / 4; 
Substrate_AvgTemp[3] := (fPV_Value_Sub[4] + fPV_Value_Sub[5] + fPV_Value_Sub[7] + fPV_Value_Sub[8]) / 4; 
Substrate_AvgTemp[4] := (fPV_Value_Sub[5] + fPV_Value_Sub[6] + fPV_Value_Sub[8] + fPV_Value_Sub[9]) / 4;
END_ACTION

ACTION Substrate_Simulation:
fMV_Out:= gbl.slave_fPV_Value;

gbl.fPV_Value_SubTC[1] := fMV_Out[1] - 2.5;
gbl.fPV_Value_SubTC[2] := (fMV_Out[1] + fMV_Out[2]) / 2 - 3.4;
gbl.fPV_Value_SubTC[3] := fMV_Out[2] - 3.1;
gbl.fPV_Value_SubTC[4] := (fMV_Out[1] + fMV_Out[3]) / 2 - 3.5;
gbl.fPV_Value_SubTC[5] := (fMV_Out[1] + fMV_Out[2]+ fMV_Out[3] + fMV_Out[4]) / 4 - 4;
gbl.fPV_Value_SubTC[6] := (fMV_Out[2] + fMV_Out[4]) / 2 - 3.2;
gbl.fPV_Value_SubTC[7] := fMV_Out[3] - 2.6;
gbl.fPV_Value_SubTC[8] := (fMV_Out[3] + fMV_Out[4]) / 2 - 3.4;
gbl.fPV_Value_SubTC[9] := fMV_Out[4] - 2.1;


(*
fMV_Out_Sub[1] := fMV_Out[1];

IF fMV_Out[1] = 0 AND fMV_Out[2] = 0 THEN
	fMV_Out_Sub[2] := 0;
ELSE
	fMV_Out_Sub[2] := (fMV_Out[1] + fMV_Out[2]) / 2;
END_IF

fMV_Out_Sub[3] := fMV_Out[2];

IF fMV_Out[1] = 0 AND fMV_Out[3] = 0 THEN
	fMV_Out_Sub[4] := 0;
ELSE
	fMV_Out_Sub[4] := (fMV_Out[1] + fMV_Out[3]) / 2;
END_IF

IF fMV_Out[1] = 0 AND fMV_Out[2] = 0 AND fMV_Out[3] = 0 AND fMV_Out[3] = 0 THEN
	fMV_Out_Sub[5] := 0;
ELSE
	fMV_Out_Sub[5] := (fMV_Out[1] + fMV_Out[2] + fMV_Out[3] + fMV_Out[4]) / 4;
END_IF

IF fMV_Out[2] = 0 AND fMV_Out[4] = 0 THEN
	fMV_Out_Sub[6] := 0;
ELSE
	fMV_Out_Sub[6] := (fMV_Out[2] + fMV_Out[4]) / 2;
END_IF

fMV_Out_Sub[7] := fMV_Out[3];

IF fMV_Out[3] = 0 AND fMV_Out[4] = 0 THEN
	fMV_Out_Sub[8] := 0;
ELSE
	fMV_Out_Sub[8] := (fMV_Out[3] + fMV_Out[4]) / 2;
END_IF

fMV_Out_Sub[9] := fMV_Out[4];


FOR i:=1 TO 9 BY 1 DO
	stPTParams_Sub[i].tTaskCycleTime	:= tTaskCycleTime;
	stPTParams_Sub[i].tCtrlCycleTime	:= tCtrlCycleTime;
	stPTParams_Sub[i].tT1				:= stPTParams_Sub[i].tT2 := tTimeConstant_Sub[i];
	stPTParams_Sub[i].fKp				:= fKp_Sub[i];


	fbCTRL_PT2_Sub[i](
					fIn			:= fMV_Out_Sub[i] ,
					eMode		:= 2,
					stParams	:= stPTParams_Sub[i],
					fOut		=> fPV_Value_Local_Sub[i]
					);	
					
	IF fPV_Value_Local_Sub[i] <= fInit_Temp_Sub[i] THEN
		fPV_Value_Sub[i] := fInit_Temp_Sub[i];
	ELSE
		fPV_Value_Sub[i] := fPV_Value_Local_Sub[i];
	END_IF 	
	
END_FOR
*)
END_ACTION

ACTION TUNING:
IF m_fTargetTemp > 0 THEN
			
	FOR i:=1 TO 4 BY 1 DO
		
		mErr_Value[i] := m_Tuning_Set_Temp[i] - Substrate_AvgTemp[i];
		mErr_integral_Val[i] := mErr_integral_Val[i] + (mErr_Value[i] * m_Sampling_Time);
		master_Zone_AVG[i] := (m_pi_gain[i] * mErr_Value[i]) + (m_pi_gain[i] / m_integral_constant[i] * mErr_integral_Val[i]) + m_Tuning_Set_Temp[i]; 
		
		m_Last_Zone_Temp_AVG[i] := master_Zone_AVG[i];
		
		IF master_Zone_AVG[i] < m_Zone_Temp_Min THEN
			master_Zone_AVG[i] := m_Zone_Temp_Min;
			mErr_integral_Val[i] :=  0;
		ELSIF master_Zone_AVG[i] > m_Zone_Temp_Max THEN
			master_Zone_AVG[i] := m_Zone_Temp_Max; 
			mErr_integral_Val[i] :=  0;
		END_IF
	END_FOR	
	gbl.slave_fTargetTemp := master_Zone_AVG;
	gbl.isChanged := TRUE;
END_IF
END_ACTION

END_PROGRAM
